(* Logix 5000 project; controller Lab6_Unit18 vendor 1 type 14 code 106 rev 30.11; software revision 30.00 *)

TASK MainTask (continuous, watchdog 500 ms) : MainProgram

MODULES
   Local : vendor 1 type 14 code 106 (Compact 0, rev 30.11)
      I1 : 1769-IQ16 (Compact 1, rev 1.1, Input RPI 20 ms)
      A3 : vendor 1 type 10 code 33 (Compact 3, rev 1.1, Output RPI 80 ms)
      O2 : vendor 1 type 7 code 86 (Compact 2, rev 2.1, Output RPI 20 ms)
END_MODULES

PROGRAM MainProgram   (* main routine MainRoutine *)
VAR
   Black_Mushroomhead_PB : ALIAS FOR Local:1:I.Data.5;
   Blue_Flush_PB : ALIAS FOR Local:1:I.Data.1;
   Blue_Indicator : ALIAS FOR Local:2:O.Data.3;
   Green_Flush_PB : ALIAS FOR Local:1:I.Data.2;
   Green_Indicator : ALIAS FOR Local:2:O.Data.1;
   Machine_Active : BOOL;
   Red_Flush_PB : ALIAS FOR Local:1:I.Data.4;
   Red_Indicator : ALIAS FOR Local:2:O.Data.5;
   Red_Mushroomhead_PB : ALIAS FOR Local:1:I.Data.6;
   White_Flush_PB : ALIAS FOR Local:1:I.Data.0;
   White_Indicator : ALIAS FOR Local:2:O.Data.4;
   Yellow_Flush_PB : ALIAS FOR Local:1:I.Data.3;
   Yellow_Indicator : ALIAS FOR Local:2:O.Data.2;
END_VAR

ROUTINE MainRoutine   (* ladder *)
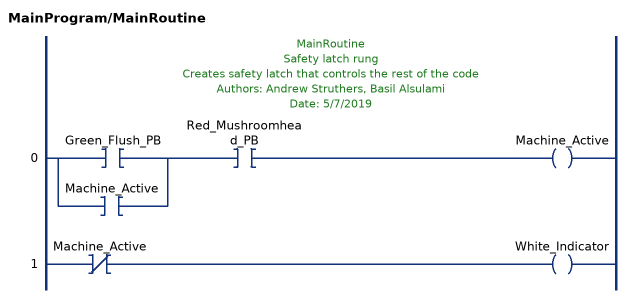
   // MainRoutine
   // Safety latch rung
   // Creates safety latch that controls the rest of the code
   // Authors: Andrew Struthers, Basil Alsulami
   // Date: 5/7/2019
   0: [XIC(Green_Flush_PB) ,XIC(Machine_Active) ]XIC(Red_Mushroomhead_PB)OTE(Machine_Active);
   1: XIO(Machine_Active)OTE(White_Indicator);
END_ROUTINE
END_PROGRAM
